// TIA Portal V18 export
FUNCTION "ER_lim_auto_ws" : Void   // FC19, FBD
{ S7_Optimized_Access := 'TRUE' }
VERSION : 0.1
// stored: AutoNumber true, IsIECCheckEnabled false, SetENOAutomatically false, UDAEnableTagReadback false
   VAR_INPUT
      par_fwd_limit : Real;
      par_rev_limit : Real;
      par_dist_fast : Real;
      par_spd_fast : Real;
      par_spd_slow : Real;
   END_VAR
   VAR_OUTPUT
      ER_settings : Bool;
      wsER : WString;
   END_VAR
   VAR_TEMP
      tmp_fwdLEREV : Bool;
      tmp_fastL0 : Bool;
      tmp_fastLEslo : Bool;
   END_VAR
BEGIN

REGION Network 1
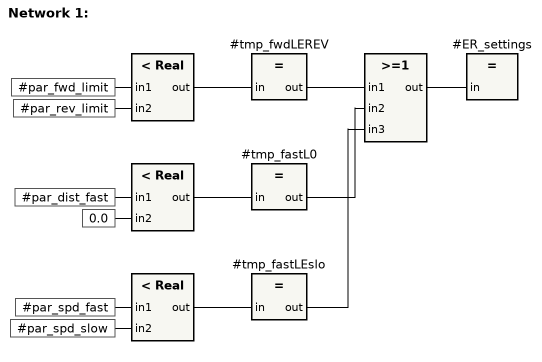
   #tmp_fwdLEREV := #par_fwd_limit < #par_rev_limit;
   #tmp_fastL0 := #par_dist_fast < 0.0;
   #tmp_fastLEslo := #par_spd_fast < #par_spd_slow;
   #ER_settings := #tmp_fwdLEREV OR #tmp_fastL0 OR #tmp_fastLEslo;
END_REGION

REGION Network 2 (SCL)
   IF #tmp_fwdLEREV THEN
       #wsER := WSTRING#'lim fwd LE rev';
   END_IF;
   IF #tmp_fastL0 THEN
       #wsER := WSTRING#'dist fast 0';
   END_IF;
   IF #tmp_fastLEslo THEN
       #wsER := WSTRING#'v fast LE slo';
   END_IF;
END_REGION
END_FUNCTION
